FUNCTION CheckDivByte : BYTE
VAR_INPUT
	divisor			 	: BYTE;
END_VAR
VAR
END_VAR

IF divisor = 0 THEN
	CheckByteZeroDiv_ErrCnt := CheckByteZeroDiv_ErrCnt + 1;
	CheckDivByte := 1;
ELSE
	CheckDivByte := divisor;
END_IF

END_FUNCTION

(* stored: Version 1.1.0.1, ProductVersion 3.1.4024.9
   POU CheckDivByte: Id {44e05fe0-f9fe-4db6-addf-2d35958f6f5c}, SpecialFunc CheckDivInt32 *)
